// Mitsubishi GX Works2 project: LRI - PLC - NOR   PLC: Q03UDV

PROGRAM MAIN
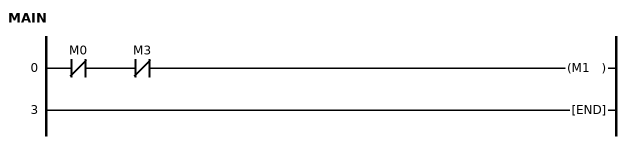
0     LDI     M0
      ANI     M3
      OUT     M1
3     END
END_PROGRAM
